(* Logix 5000 project; controller UnitTest_Controller 1756-L85E rev 36.11; software revision 36.00 *)

TASK T00_UnitTesting (continuous, watchdog 500 ms) : P00_UnitTesting

MODULES
   Local : 1756-L85E (ICP 0, rev 36.11)
END_MODULES

TYPE FAULTRECORD :
STRUCT
   Time_Low : DINT;   // Lower 32 bits of the fault timestamp value
   Time_High : DINT;   // Upper 32 bits of the fault timestamp value
   Type : INT;   // Fault type (program, I/O, and so forth)
   Code : INT;   // Unique code for the fault
   Info : DINT[8];   // Fault specific information
END_STRUCT
END_TYPE

ADD_ON_INSTRUCTION RectAreaCalcAndCompare   (* revision 1.0 *)
VAR_INPUT
   box_length : SINT; {required}
   box_width : DINT; {required}
   compareValue_for_box_Area : DINT; {required}
END_VAR
VAR_OUTPUT
   box_area : LINT; {access Read Only, required}
   area_comparison_result : BOOL; {access Read Only, visible}
END_VAR

ROUTINE Logic   (* ladder *)
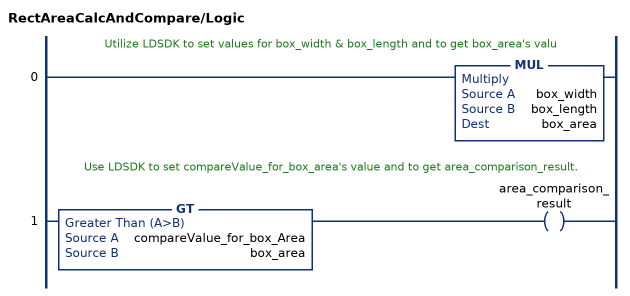
   // Utilize LDSDK to set values for box_width & box_length and to get box_area's valu
   0: MUL(box_width,box_length,box_area);
   // Use LDSDK to set compareValue_for_box_area's value and to get area_comparison_result.
   1: GT(compareValue_for_box_Area,box_area)OTE(area_comparison_result);
END_ROUTINE
END_ADD_ON_INSTRUCTION

VAR_GLOBAL   (* controller tags *)
   AOI_RectAreaCalcAndCompare : RectAreaCalcAndCompare;   // Automated Testing -------------------- generated AOI tag being unit tested
   AT_ClearFault : BOOL;   // Automated Testing -------------------- clear the fault type & code
   AT_EnableIn : BOOL;   // Automated Testing -------------------- set the EnableIn AOI input parameter
   AT_FaultCode : DINT;   // Automated Testing -------------------- contains fault code number
   AT_FaultedIndicator : BOOL;   // Automated Testing -------------------- boolean HIGH if controller faulted
   AT_FaultType : DINT;   // Automated Testing -------------------- contains fault type number
   AT_ToggleTest : BOOL;   // Automated Testing -------------------- toggle to progress AOI testing by 1 clock cycle
   major_fault_record : FAULTRECORD;
   ONS : BOOL;   // Automated Testing -------------------- make the routine with AOI being tested update only 1 clock cycle
END_VAR

PROGRAM P00_UnitTesting   (* main routine R00_MainRoutine *)

ROUTINE R00_MainRoutine   (* ladder *)
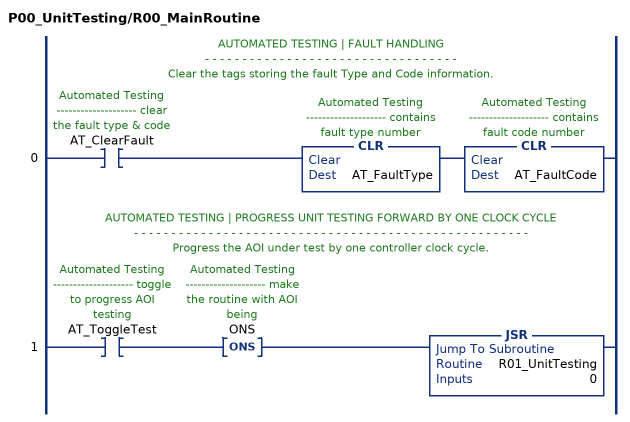
   // AUTOMATED TESTING | FAULT HANDLING
   // - - - - - - - - - - - - - - - - - - - - - - - - - - - - - - - - - -
   // Clear the tags storing the fault Type and Code information.
   0: XIC(AT_ClearFault)CLR(AT_FaultType)CLR(AT_FaultCode);
   // AUTOMATED TESTING | PROGRESS UNIT TESTING FORWARD BY ONE CLOCK CYCLE
   // - - - - - - - - - - - - - - - - - - - - - - - - - - - - - - - - - - - - - - - - - - - - - - - - - - - - -
   // Progress the AOI under test by one controller clock cycle.
   1: XIC(AT_ToggleTest)ONS(ONS)JSR(R01_UnitTesting,0);
END_ROUTINE

ROUTINE R01_UnitTesting   (* ladder *)
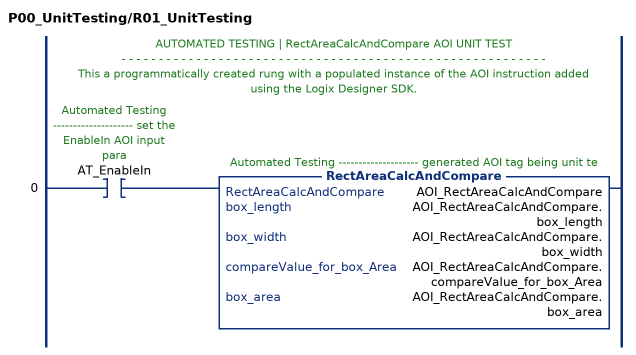
   // AUTOMATED TESTING | RectAreaCalcAndCompare AOI UNIT TEST
   // - - - - - - - - - - - - - - - - - - - - - - - - - - - - - - - - - - - - - - - - - - - - - - - - - - - - - - - - -
   // This a programmatically created rung with a populated instance of the AOI instruction added using the Logix Designer SDK.
   0: XIC(AT_EnableIn)RectAreaCalcAndCompare(AOI_RectAreaCalcAndCompare,AOI_RectAreaCalcAndCompare.box_length,AOI_RectAreaCalcAndCompare.box_width,AOI_RectAreaCalcAndCompare.compareValue_for_box_Area,AOI_RectAreaCalcAndCompare.box_area);
END_ROUTINE
END_PROGRAM

PROGRAM PXX_FaultHandler   (* main routine RXX_FaultHandler *)

ROUTINE RXX_FaultHandler   (* ladder *)
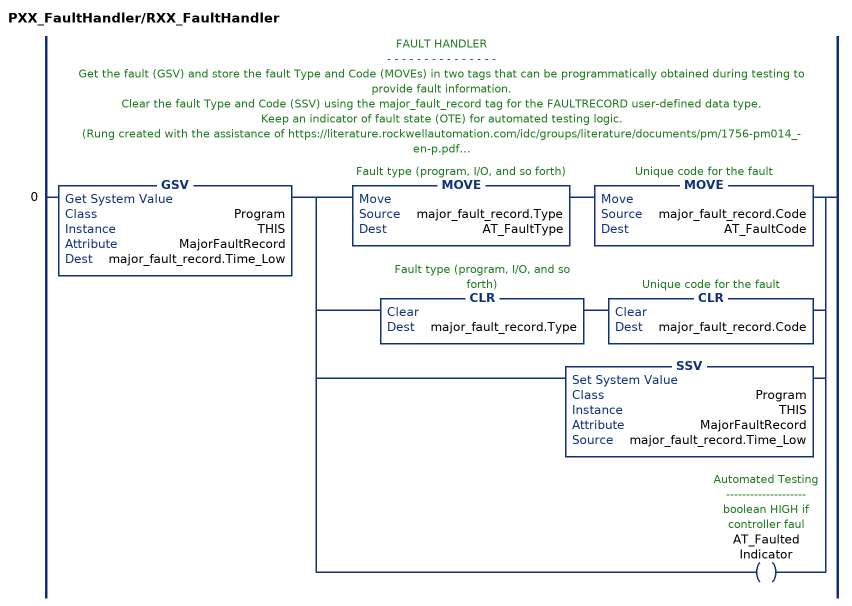
   // FAULT HANDLER
   // - - - - - - - - - - - - - - -
   // Get the fault (GSV) and store the fault Type and Code (MOVEs) in two tags that can be programmatically obtained during testing to provide fault information.
   // Clear the fault Type and Code (SSV) using the major_fault_record tag for the FAULTRECORD user-defined data type.
   // Keep an indicator of fault state (OTE) for automated testing logic.
   // (Rung created with the assistance of https://literature.rockwellautomation.com/idc/groups/literature/documents/pm/1756-pm014_-en-p.pdf)
   // (Fault code spreadsheet link: https://literature.rockwellautomation.com/idc/groups/literature/documents/rd/1756-rd001_-en-p.xlsx)
   0: GSV(Program,THIS,MajorFaultRecord,major_fault_record.Time_Low)[MOVE(major_fault_record.Type,AT_FaultType) MOVE(major_fault_record.Code,AT_FaultCode) ,CLR(major_fault_record.Type) CLR(major_fault_record.Code) ,SSV(Program,THIS,MajorFaultRecord,major_fault_record.Time_Low) ,OTE(AT_FaultedIndicator) ];
END_ROUTINE
END_PROGRAM
